// TIA Portal V18 export
FUNCTION "SS1_A6_16DI_IO_Update" : Void   // FC11060, LAD
{ S7_Optimized_Access := 'TRUE' }
VERSION : 0.1
// stored: AutoNumber false, IsIECCheckEnabled false, SetENOAutomatically false, UDAEnableTagReadback false
BEGIN

REGION Network 1: DIa0
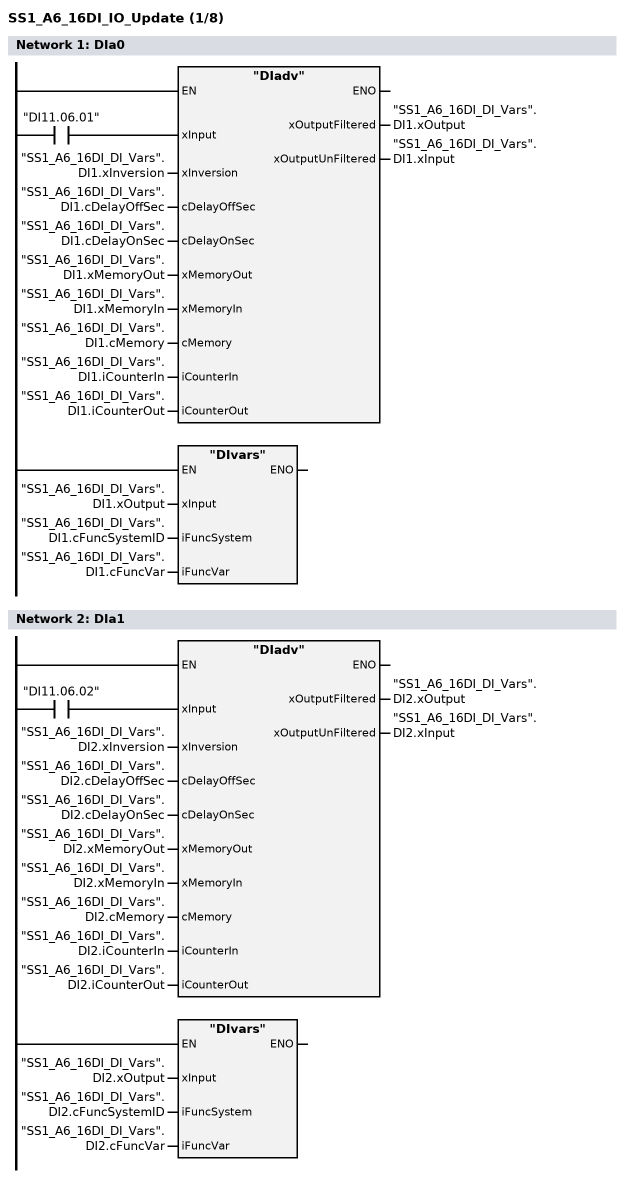
   RUNG wire#powerrail
      "DIadv"(xInput := wire#w1, xInversion := "SS1_A6_16DI_DI_Vars".DI1.xInversion, cDelayOffSec := "SS1_A6_16DI_DI_Vars".DI1.cDelayOffSec, cDelayOnSec := "SS1_A6_16DI_DI_Vars".DI1.cDelayOnSec, xMemoryOut := "SS1_A6_16DI_DI_Vars".DI1.xMemoryOut, xMemoryIn := "SS1_A6_16DI_DI_Vars".DI1.xMemoryIn, cMemory := "SS1_A6_16DI_DI_Vars".DI1.cMemory, xOutputFiltered => "SS1_A6_16DI_DI_Vars".DI1.xOutput, xOutputUnFiltered => "SS1_A6_16DI_DI_Vars".DI1.xInput, iCounterIn := "SS1_A6_16DI_DI_Vars".DI1.iCounterIn, iCounterOut := "SS1_A6_16DI_DI_Vars".DI1.iCounterOut)
   END_RUNG
   RUNG wire#powerrail
      Contact( "DI11.06.01" )
   END_RUNG wire#w1
   RUNG wire#powerrail
      "DIvars"(xInput := "SS1_A6_16DI_DI_Vars".DI1.xOutput, iFuncSystem := "SS1_A6_16DI_DI_Vars".DI1.cFuncSystemID, iFuncVar := "SS1_A6_16DI_DI_Vars".DI1.cFuncVar)
   END_RUNG
   // the same network as SCL:
   "DIadv"(xInput := "DI11.06.01",
           xInversion := "SS1_A6_16DI_DI_Vars".DI1.xInversion,
           cDelayOffSec := "SS1_A6_16DI_DI_Vars".DI1.cDelayOffSec,
           cDelayOnSec := "SS1_A6_16DI_DI_Vars".DI1.cDelayOnSec,
           xMemoryOut := "SS1_A6_16DI_DI_Vars".DI1.xMemoryOut,
           xMemoryIn := "SS1_A6_16DI_DI_Vars".DI1.xMemoryIn,
           cMemory := "SS1_A6_16DI_DI_Vars".DI1.cMemory,
           iCounterIn := "SS1_A6_16DI_DI_Vars".DI1.iCounterIn,
           iCounterOut := "SS1_A6_16DI_DI_Vars".DI1.iCounterOut,
           xOutputFiltered => "SS1_A6_16DI_DI_Vars".DI1.xOutput,
           xOutputUnFiltered => "SS1_A6_16DI_DI_Vars".DI1.xInput);
   "DIvars"(xInput := "SS1_A6_16DI_DI_Vars".DI1.xOutput,
            iFuncSystem := "SS1_A6_16DI_DI_Vars".DI1.cFuncSystemID,
            iFuncVar := "SS1_A6_16DI_DI_Vars".DI1.cFuncVar);
END_REGION

REGION Network 2: DIa1
   RUNG wire#powerrail
      "DIadv"(xInput := wire#w1, xInversion := "SS1_A6_16DI_DI_Vars".DI2.xInversion, cDelayOffSec := "SS1_A6_16DI_DI_Vars".DI2.cDelayOffSec, cDelayOnSec := "SS1_A6_16DI_DI_Vars".DI2.cDelayOnSec, xMemoryOut := "SS1_A6_16DI_DI_Vars".DI2.xMemoryOut, xMemoryIn := "SS1_A6_16DI_DI_Vars".DI2.xMemoryIn, cMemory := "SS1_A6_16DI_DI_Vars".DI2.cMemory, xOutputFiltered => "SS1_A6_16DI_DI_Vars".DI2.xOutput, xOutputUnFiltered => "SS1_A6_16DI_DI_Vars".DI2.xInput, iCounterIn := "SS1_A6_16DI_DI_Vars".DI2.iCounterIn, iCounterOut := "SS1_A6_16DI_DI_Vars".DI2.iCounterOut)
   END_RUNG
   RUNG wire#powerrail
      Contact( "DI11.06.02" )
   END_RUNG wire#w1
   RUNG wire#powerrail
      "DIvars"(xInput := "SS1_A6_16DI_DI_Vars".DI2.xOutput, iFuncSystem := "SS1_A6_16DI_DI_Vars".DI2.cFuncSystemID, iFuncVar := "SS1_A6_16DI_DI_Vars".DI2.cFuncVar)
   END_RUNG
   // the same network as SCL:
   "DIadv"(xInput := "DI11.06.02",
           xInversion := "SS1_A6_16DI_DI_Vars".DI2.xInversion,
           cDelayOffSec := "SS1_A6_16DI_DI_Vars".DI2.cDelayOffSec,
           cDelayOnSec := "SS1_A6_16DI_DI_Vars".DI2.cDelayOnSec,
           xMemoryOut := "SS1_A6_16DI_DI_Vars".DI2.xMemoryOut,
           xMemoryIn := "SS1_A6_16DI_DI_Vars".DI2.xMemoryIn,
           cMemory := "SS1_A6_16DI_DI_Vars".DI2.cMemory,
           iCounterIn := "SS1_A6_16DI_DI_Vars".DI2.iCounterIn,
           iCounterOut := "SS1_A6_16DI_DI_Vars".DI2.iCounterOut,
           xOutputFiltered => "SS1_A6_16DI_DI_Vars".DI2.xOutput,
           xOutputUnFiltered => "SS1_A6_16DI_DI_Vars".DI2.xInput);
   "DIvars"(xInput := "SS1_A6_16DI_DI_Vars".DI2.xOutput,
            iFuncSystem := "SS1_A6_16DI_DI_Vars".DI2.cFuncSystemID,
            iFuncVar := "SS1_A6_16DI_DI_Vars".DI2.cFuncVar);
END_REGION

REGION Network 3: DIa2
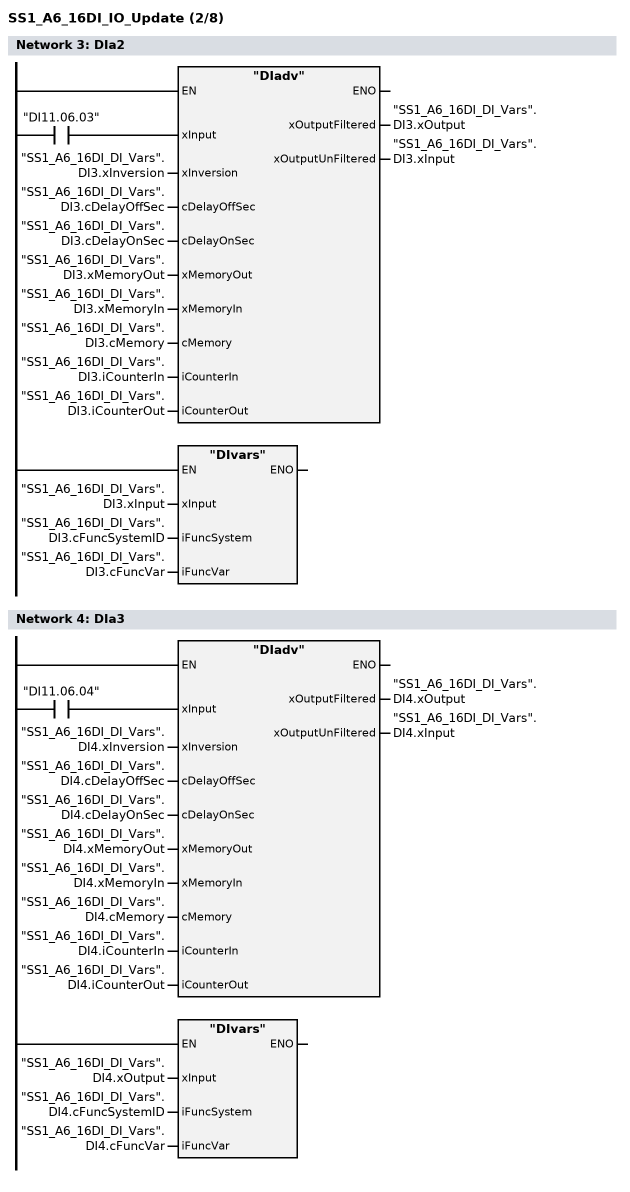
   RUNG wire#powerrail
      "DIadv"(xInput := wire#w1, xInversion := "SS1_A6_16DI_DI_Vars".DI3.xInversion, cDelayOffSec := "SS1_A6_16DI_DI_Vars".DI3.cDelayOffSec, cDelayOnSec := "SS1_A6_16DI_DI_Vars".DI3.cDelayOnSec, xMemoryOut := "SS1_A6_16DI_DI_Vars".DI3.xMemoryOut, xMemoryIn := "SS1_A6_16DI_DI_Vars".DI3.xMemoryIn, cMemory := "SS1_A6_16DI_DI_Vars".DI3.cMemory, xOutputFiltered => "SS1_A6_16DI_DI_Vars".DI3.xOutput, xOutputUnFiltered => "SS1_A6_16DI_DI_Vars".DI3.xInput, iCounterIn := "SS1_A6_16DI_DI_Vars".DI3.iCounterIn, iCounterOut := "SS1_A6_16DI_DI_Vars".DI3.iCounterOut)
   END_RUNG
   RUNG wire#powerrail
      Contact( "DI11.06.03" )
   END_RUNG wire#w1
   RUNG wire#powerrail
      "DIvars"(xInput := "SS1_A6_16DI_DI_Vars".DI3.xInput, iFuncSystem := "SS1_A6_16DI_DI_Vars".DI3.cFuncSystemID, iFuncVar := "SS1_A6_16DI_DI_Vars".DI3.cFuncVar)
   END_RUNG
   // the same network as SCL:
   "DIadv"(xInput := "DI11.06.03",
           xInversion := "SS1_A6_16DI_DI_Vars".DI3.xInversion,
           cDelayOffSec := "SS1_A6_16DI_DI_Vars".DI3.cDelayOffSec,
           cDelayOnSec := "SS1_A6_16DI_DI_Vars".DI3.cDelayOnSec,
           xMemoryOut := "SS1_A6_16DI_DI_Vars".DI3.xMemoryOut,
           xMemoryIn := "SS1_A6_16DI_DI_Vars".DI3.xMemoryIn,
           cMemory := "SS1_A6_16DI_DI_Vars".DI3.cMemory,
           iCounterIn := "SS1_A6_16DI_DI_Vars".DI3.iCounterIn,
           iCounterOut := "SS1_A6_16DI_DI_Vars".DI3.iCounterOut,
           xOutputFiltered => "SS1_A6_16DI_DI_Vars".DI3.xOutput,
           xOutputUnFiltered => "SS1_A6_16DI_DI_Vars".DI3.xInput);
   "DIvars"(xInput := "SS1_A6_16DI_DI_Vars".DI3.xInput,
            iFuncSystem := "SS1_A6_16DI_DI_Vars".DI3.cFuncSystemID,
            iFuncVar := "SS1_A6_16DI_DI_Vars".DI3.cFuncVar);
END_REGION

REGION Network 4: DIa3
   RUNG wire#powerrail
      "DIadv"(xInput := wire#w1, xInversion := "SS1_A6_16DI_DI_Vars".DI4.xInversion, cDelayOffSec := "SS1_A6_16DI_DI_Vars".DI4.cDelayOffSec, cDelayOnSec := "SS1_A6_16DI_DI_Vars".DI4.cDelayOnSec, xMemoryOut := "SS1_A6_16DI_DI_Vars".DI4.xMemoryOut, xMemoryIn := "SS1_A6_16DI_DI_Vars".DI4.xMemoryIn, cMemory := "SS1_A6_16DI_DI_Vars".DI4.cMemory, xOutputFiltered => "SS1_A6_16DI_DI_Vars".DI4.xOutput, xOutputUnFiltered => "SS1_A6_16DI_DI_Vars".DI4.xInput, iCounterIn := "SS1_A6_16DI_DI_Vars".DI4.iCounterIn, iCounterOut := "SS1_A6_16DI_DI_Vars".DI4.iCounterOut)
   END_RUNG
   RUNG wire#powerrail
      Contact( "DI11.06.04" )
   END_RUNG wire#w1
   RUNG wire#powerrail
      "DIvars"(xInput := "SS1_A6_16DI_DI_Vars".DI4.xOutput, iFuncSystem := "SS1_A6_16DI_DI_Vars".DI4.cFuncSystemID, iFuncVar := "SS1_A6_16DI_DI_Vars".DI4.cFuncVar)
   END_RUNG
   // the same network as SCL:
   "DIadv"(xInput := "DI11.06.04",
           xInversion := "SS1_A6_16DI_DI_Vars".DI4.xInversion,
           cDelayOffSec := "SS1_A6_16DI_DI_Vars".DI4.cDelayOffSec,
           cDelayOnSec := "SS1_A6_16DI_DI_Vars".DI4.cDelayOnSec,
           xMemoryOut := "SS1_A6_16DI_DI_Vars".DI4.xMemoryOut,
           xMemoryIn := "SS1_A6_16DI_DI_Vars".DI4.xMemoryIn,
           cMemory := "SS1_A6_16DI_DI_Vars".DI4.cMemory,
           iCounterIn := "SS1_A6_16DI_DI_Vars".DI4.iCounterIn,
           iCounterOut := "SS1_A6_16DI_DI_Vars".DI4.iCounterOut,
           xOutputFiltered => "SS1_A6_16DI_DI_Vars".DI4.xOutput,
           xOutputUnFiltered => "SS1_A6_16DI_DI_Vars".DI4.xInput);
   "DIvars"(xInput := "SS1_A6_16DI_DI_Vars".DI4.xOutput,
            iFuncSystem := "SS1_A6_16DI_DI_Vars".DI4.cFuncSystemID,
            iFuncVar := "SS1_A6_16DI_DI_Vars".DI4.cFuncVar);
END_REGION

REGION Network 5: DIa4
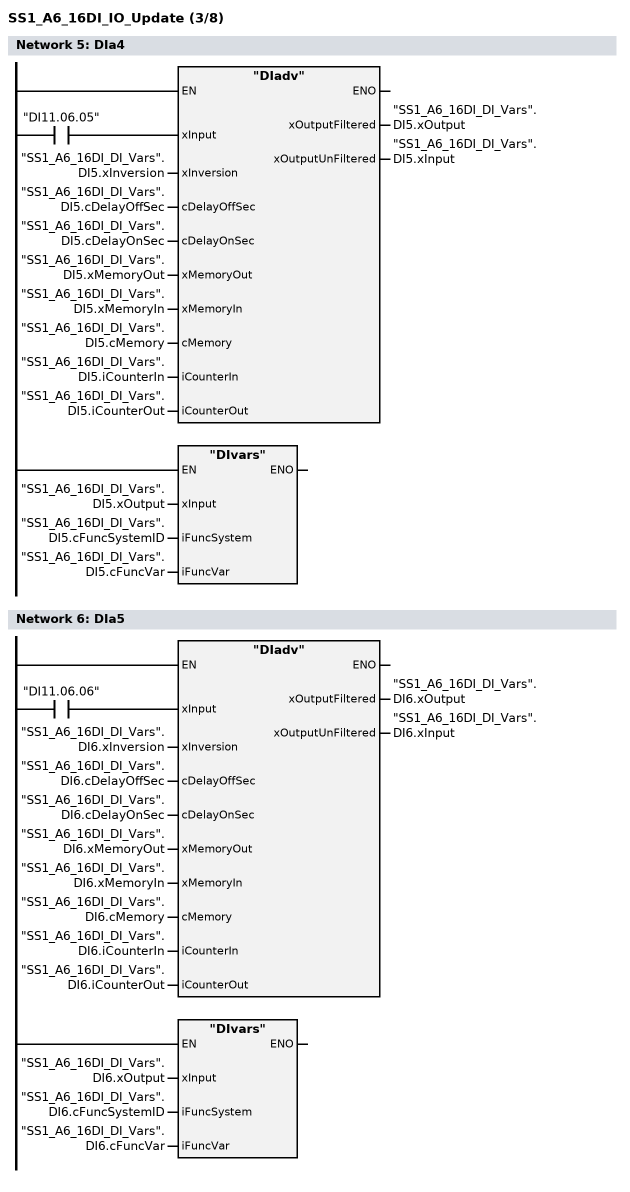
   RUNG wire#powerrail
      "DIadv"(xInput := wire#w1, xInversion := "SS1_A6_16DI_DI_Vars".DI5.xInversion, cDelayOffSec := "SS1_A6_16DI_DI_Vars".DI5.cDelayOffSec, cDelayOnSec := "SS1_A6_16DI_DI_Vars".DI5.cDelayOnSec, xMemoryOut := "SS1_A6_16DI_DI_Vars".DI5.xMemoryOut, xMemoryIn := "SS1_A6_16DI_DI_Vars".DI5.xMemoryIn, cMemory := "SS1_A6_16DI_DI_Vars".DI5.cMemory, xOutputFiltered => "SS1_A6_16DI_DI_Vars".DI5.xOutput, xOutputUnFiltered => "SS1_A6_16DI_DI_Vars".DI5.xInput, iCounterIn := "SS1_A6_16DI_DI_Vars".DI5.iCounterIn, iCounterOut := "SS1_A6_16DI_DI_Vars".DI5.iCounterOut)
   END_RUNG
   RUNG wire#powerrail
      Contact( "DI11.06.05" )
   END_RUNG wire#w1
   RUNG wire#powerrail
      "DIvars"(xInput := "SS1_A6_16DI_DI_Vars".DI5.xOutput, iFuncSystem := "SS1_A6_16DI_DI_Vars".DI5.cFuncSystemID, iFuncVar := "SS1_A6_16DI_DI_Vars".DI5.cFuncVar)
   END_RUNG
   // the same network as SCL:
   "DIadv"(xInput := "DI11.06.05",
           xInversion := "SS1_A6_16DI_DI_Vars".DI5.xInversion,
           cDelayOffSec := "SS1_A6_16DI_DI_Vars".DI5.cDelayOffSec,
           cDelayOnSec := "SS1_A6_16DI_DI_Vars".DI5.cDelayOnSec,
           xMemoryOut := "SS1_A6_16DI_DI_Vars".DI5.xMemoryOut,
           xMemoryIn := "SS1_A6_16DI_DI_Vars".DI5.xMemoryIn,
           cMemory := "SS1_A6_16DI_DI_Vars".DI5.cMemory,
           iCounterIn := "SS1_A6_16DI_DI_Vars".DI5.iCounterIn,
           iCounterOut := "SS1_A6_16DI_DI_Vars".DI5.iCounterOut,
           xOutputFiltered => "SS1_A6_16DI_DI_Vars".DI5.xOutput,
           xOutputUnFiltered => "SS1_A6_16DI_DI_Vars".DI5.xInput);
   "DIvars"(xInput := "SS1_A6_16DI_DI_Vars".DI5.xOutput,
            iFuncSystem := "SS1_A6_16DI_DI_Vars".DI5.cFuncSystemID,
            iFuncVar := "SS1_A6_16DI_DI_Vars".DI5.cFuncVar);
END_REGION

REGION Network 6: DIa5
   RUNG wire#powerrail
      "DIadv"(xInput := wire#w1, xInversion := "SS1_A6_16DI_DI_Vars".DI6.xInversion, cDelayOffSec := "SS1_A6_16DI_DI_Vars".DI6.cDelayOffSec, cDelayOnSec := "SS1_A6_16DI_DI_Vars".DI6.cDelayOnSec, xMemoryOut := "SS1_A6_16DI_DI_Vars".DI6.xMemoryOut, xMemoryIn := "SS1_A6_16DI_DI_Vars".DI6.xMemoryIn, cMemory := "SS1_A6_16DI_DI_Vars".DI6.cMemory, xOutputFiltered => "SS1_A6_16DI_DI_Vars".DI6.xOutput, xOutputUnFiltered => "SS1_A6_16DI_DI_Vars".DI6.xInput, iCounterIn := "SS1_A6_16DI_DI_Vars".DI6.iCounterIn, iCounterOut := "SS1_A6_16DI_DI_Vars".DI6.iCounterOut)
   END_RUNG
   RUNG wire#powerrail
      Contact( "DI11.06.06" )
   END_RUNG wire#w1
   RUNG wire#powerrail
      "DIvars"(xInput := "SS1_A6_16DI_DI_Vars".DI6.xOutput, iFuncSystem := "SS1_A6_16DI_DI_Vars".DI6.cFuncSystemID, iFuncVar := "SS1_A6_16DI_DI_Vars".DI6.cFuncVar)
   END_RUNG
   // the same network as SCL:
   "DIadv"(xInput := "DI11.06.06",
           xInversion := "SS1_A6_16DI_DI_Vars".DI6.xInversion,
           cDelayOffSec := "SS1_A6_16DI_DI_Vars".DI6.cDelayOffSec,
           cDelayOnSec := "SS1_A6_16DI_DI_Vars".DI6.cDelayOnSec,
           xMemoryOut := "SS1_A6_16DI_DI_Vars".DI6.xMemoryOut,
           xMemoryIn := "SS1_A6_16DI_DI_Vars".DI6.xMemoryIn,
           cMemory := "SS1_A6_16DI_DI_Vars".DI6.cMemory,
           iCounterIn := "SS1_A6_16DI_DI_Vars".DI6.iCounterIn,
           iCounterOut := "SS1_A6_16DI_DI_Vars".DI6.iCounterOut,
           xOutputFiltered => "SS1_A6_16DI_DI_Vars".DI6.xOutput,
           xOutputUnFiltered => "SS1_A6_16DI_DI_Vars".DI6.xInput);
   "DIvars"(xInput := "SS1_A6_16DI_DI_Vars".DI6.xOutput,
            iFuncSystem := "SS1_A6_16DI_DI_Vars".DI6.cFuncSystemID,
            iFuncVar := "SS1_A6_16DI_DI_Vars".DI6.cFuncVar);
END_REGION

REGION Network 7: DIa6
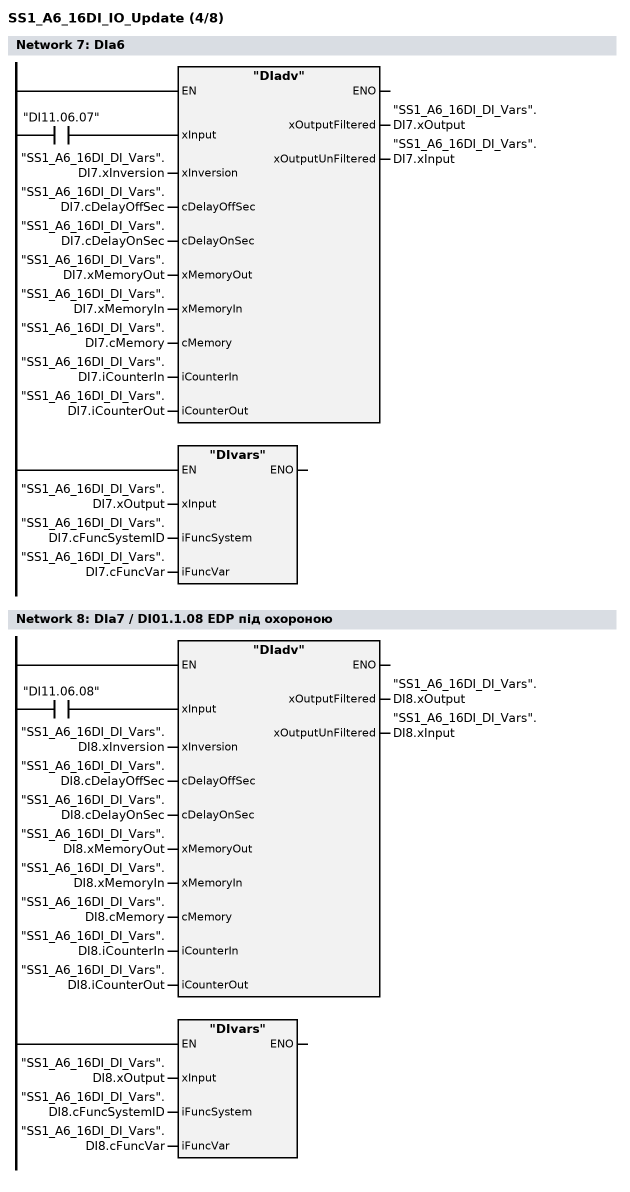
   RUNG wire#powerrail
      "DIadv"(xInput := wire#w1, xInversion := "SS1_A6_16DI_DI_Vars".DI7.xInversion, cDelayOffSec := "SS1_A6_16DI_DI_Vars".DI7.cDelayOffSec, cDelayOnSec := "SS1_A6_16DI_DI_Vars".DI7.cDelayOnSec, xMemoryOut := "SS1_A6_16DI_DI_Vars".DI7.xMemoryOut, xMemoryIn := "SS1_A6_16DI_DI_Vars".DI7.xMemoryIn, cMemory := "SS1_A6_16DI_DI_Vars".DI7.cMemory, xOutputFiltered => "SS1_A6_16DI_DI_Vars".DI7.xOutput, xOutputUnFiltered => "SS1_A6_16DI_DI_Vars".DI7.xInput, iCounterIn := "SS1_A6_16DI_DI_Vars".DI7.iCounterIn, iCounterOut := "SS1_A6_16DI_DI_Vars".DI7.iCounterOut)
   END_RUNG
   RUNG wire#powerrail
      Contact( "DI11.06.07" )
   END_RUNG wire#w1
   RUNG wire#powerrail
      "DIvars"(xInput := "SS1_A6_16DI_DI_Vars".DI7.xOutput, iFuncSystem := "SS1_A6_16DI_DI_Vars".DI7.cFuncSystemID, iFuncVar := "SS1_A6_16DI_DI_Vars".DI7.cFuncVar)
   END_RUNG
   // the same network as SCL:
   "DIadv"(xInput := "DI11.06.07",
           xInversion := "SS1_A6_16DI_DI_Vars".DI7.xInversion,
           cDelayOffSec := "SS1_A6_16DI_DI_Vars".DI7.cDelayOffSec,
           cDelayOnSec := "SS1_A6_16DI_DI_Vars".DI7.cDelayOnSec,
           xMemoryOut := "SS1_A6_16DI_DI_Vars".DI7.xMemoryOut,
           xMemoryIn := "SS1_A6_16DI_DI_Vars".DI7.xMemoryIn,
           cMemory := "SS1_A6_16DI_DI_Vars".DI7.cMemory,
           iCounterIn := "SS1_A6_16DI_DI_Vars".DI7.iCounterIn,
           iCounterOut := "SS1_A6_16DI_DI_Vars".DI7.iCounterOut,
           xOutputFiltered => "SS1_A6_16DI_DI_Vars".DI7.xOutput,
           xOutputUnFiltered => "SS1_A6_16DI_DI_Vars".DI7.xInput);
   "DIvars"(xInput := "SS1_A6_16DI_DI_Vars".DI7.xOutput,
            iFuncSystem := "SS1_A6_16DI_DI_Vars".DI7.cFuncSystemID,
            iFuncVar := "SS1_A6_16DI_DI_Vars".DI7.cFuncVar);
END_REGION

REGION Network 8: DIa7 / DI01.1.08 EDP під охороною
   RUNG wire#powerrail
      "DIadv"(xInput := wire#w1, xInversion := "SS1_A6_16DI_DI_Vars".DI8.xInversion, cDelayOffSec := "SS1_A6_16DI_DI_Vars".DI8.cDelayOffSec, cDelayOnSec := "SS1_A6_16DI_DI_Vars".DI8.cDelayOnSec, xMemoryOut := "SS1_A6_16DI_DI_Vars".DI8.xMemoryOut, xMemoryIn := "SS1_A6_16DI_DI_Vars".DI8.xMemoryIn, cMemory := "SS1_A6_16DI_DI_Vars".DI8.cMemory, xOutputFiltered => "SS1_A6_16DI_DI_Vars".DI8.xOutput, xOutputUnFiltered => "SS1_A6_16DI_DI_Vars".DI8.xInput, iCounterIn := "SS1_A6_16DI_DI_Vars".DI8.iCounterIn, iCounterOut := "SS1_A6_16DI_DI_Vars".DI8.iCounterOut)
   END_RUNG
   RUNG wire#powerrail
      Contact( "DI11.06.08" )
   END_RUNG wire#w1
   RUNG wire#powerrail
      "DIvars"(xInput := "SS1_A6_16DI_DI_Vars".DI8.xOutput, iFuncSystem := "SS1_A6_16DI_DI_Vars".DI8.cFuncSystemID, iFuncVar := "SS1_A6_16DI_DI_Vars".DI8.cFuncVar)
   END_RUNG
   // the same network as SCL:
   "DIadv"(xInput := "DI11.06.08",
           xInversion := "SS1_A6_16DI_DI_Vars".DI8.xInversion,
           cDelayOffSec := "SS1_A6_16DI_DI_Vars".DI8.cDelayOffSec,
           cDelayOnSec := "SS1_A6_16DI_DI_Vars".DI8.cDelayOnSec,
           xMemoryOut := "SS1_A6_16DI_DI_Vars".DI8.xMemoryOut,
           xMemoryIn := "SS1_A6_16DI_DI_Vars".DI8.xMemoryIn,
           cMemory := "SS1_A6_16DI_DI_Vars".DI8.cMemory,
           iCounterIn := "SS1_A6_16DI_DI_Vars".DI8.iCounterIn,
           iCounterOut := "SS1_A6_16DI_DI_Vars".DI8.iCounterOut,
           xOutputFiltered => "SS1_A6_16DI_DI_Vars".DI8.xOutput,
           xOutputUnFiltered => "SS1_A6_16DI_DI_Vars".DI8.xInput);
   "DIvars"(xInput := "SS1_A6_16DI_DI_Vars".DI8.xOutput,
            iFuncSystem := "SS1_A6_16DI_DI_Vars".DI8.cFuncSystemID,
            iFuncVar := "SS1_A6_16DI_DI_Vars".DI8.cFuncVar);
END_REGION

REGION Network 9: DIb0
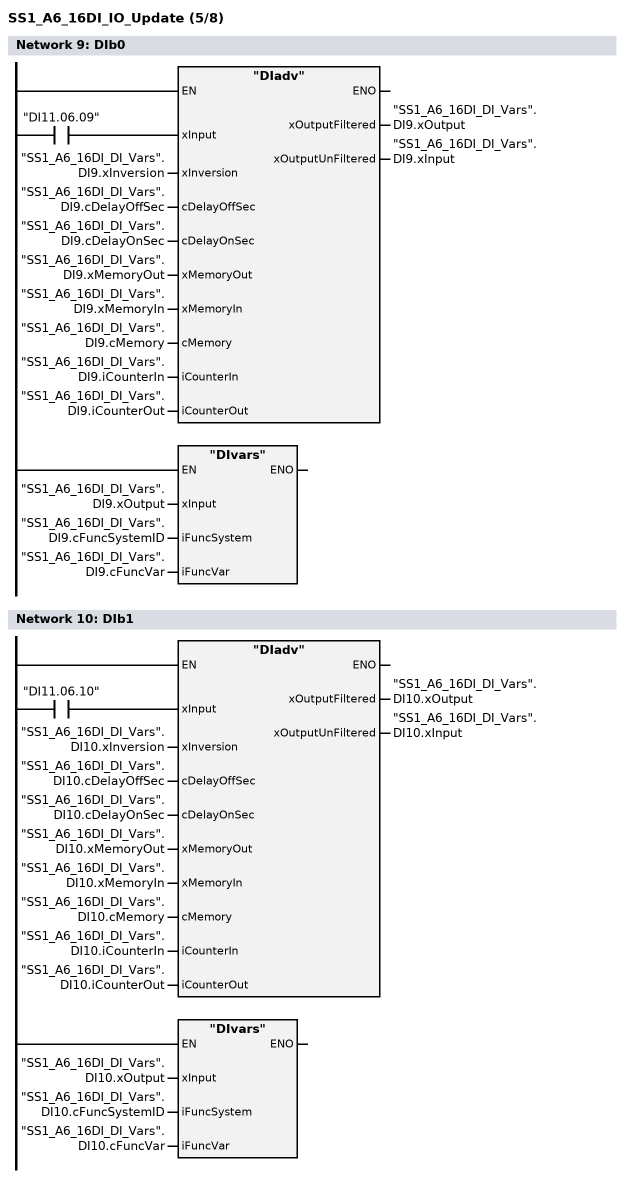
   RUNG wire#powerrail
      "DIadv"(xInput := wire#w1, xInversion := "SS1_A6_16DI_DI_Vars".DI9.xInversion, cDelayOffSec := "SS1_A6_16DI_DI_Vars".DI9.cDelayOffSec, cDelayOnSec := "SS1_A6_16DI_DI_Vars".DI9.cDelayOnSec, xMemoryOut := "SS1_A6_16DI_DI_Vars".DI9.xMemoryOut, xMemoryIn := "SS1_A6_16DI_DI_Vars".DI9.xMemoryIn, cMemory := "SS1_A6_16DI_DI_Vars".DI9.cMemory, iCounterIn := "SS1_A6_16DI_DI_Vars".DI9.iCounterIn, iCounterOut := "SS1_A6_16DI_DI_Vars".DI9.iCounterOut, xOutputFiltered => "SS1_A6_16DI_DI_Vars".DI9.xOutput, xOutputUnFiltered => "SS1_A6_16DI_DI_Vars".DI9.xInput)
   END_RUNG
   RUNG wire#powerrail
      Contact( "DI11.06.09" )
   END_RUNG wire#w1
   RUNG wire#powerrail
      "DIvars"(xInput := "SS1_A6_16DI_DI_Vars".DI9.xOutput, iFuncSystem := "SS1_A6_16DI_DI_Vars".DI9.cFuncSystemID, iFuncVar := "SS1_A6_16DI_DI_Vars".DI9.cFuncVar)
   END_RUNG
   // the same network as SCL:
   "DIadv"(xInput := "DI11.06.09",
           xInversion := "SS1_A6_16DI_DI_Vars".DI9.xInversion,
           cDelayOffSec := "SS1_A6_16DI_DI_Vars".DI9.cDelayOffSec,
           cDelayOnSec := "SS1_A6_16DI_DI_Vars".DI9.cDelayOnSec,
           xMemoryOut := "SS1_A6_16DI_DI_Vars".DI9.xMemoryOut,
           xMemoryIn := "SS1_A6_16DI_DI_Vars".DI9.xMemoryIn,
           cMemory := "SS1_A6_16DI_DI_Vars".DI9.cMemory,
           iCounterIn := "SS1_A6_16DI_DI_Vars".DI9.iCounterIn,
           iCounterOut := "SS1_A6_16DI_DI_Vars".DI9.iCounterOut,
           xOutputFiltered => "SS1_A6_16DI_DI_Vars".DI9.xOutput,
           xOutputUnFiltered => "SS1_A6_16DI_DI_Vars".DI9.xInput);
   "DIvars"(xInput := "SS1_A6_16DI_DI_Vars".DI9.xOutput,
            iFuncSystem := "SS1_A6_16DI_DI_Vars".DI9.cFuncSystemID,
            iFuncVar := "SS1_A6_16DI_DI_Vars".DI9.cFuncVar);
END_REGION

REGION Network 10: DIb1
   RUNG wire#powerrail
      "DIadv"(xInput := wire#w1, xInversion := "SS1_A6_16DI_DI_Vars".DI10.xInversion, cDelayOffSec := "SS1_A6_16DI_DI_Vars".DI10.cDelayOffSec, cDelayOnSec := "SS1_A6_16DI_DI_Vars".DI10.cDelayOnSec, xMemoryOut := "SS1_A6_16DI_DI_Vars".DI10.xMemoryOut, xMemoryIn := "SS1_A6_16DI_DI_Vars".DI10.xMemoryIn, cMemory := "SS1_A6_16DI_DI_Vars".DI10.cMemory, iCounterIn := "SS1_A6_16DI_DI_Vars".DI10.iCounterIn, iCounterOut := "SS1_A6_16DI_DI_Vars".DI10.iCounterOut, xOutputFiltered => "SS1_A6_16DI_DI_Vars".DI10.xOutput, xOutputUnFiltered => "SS1_A6_16DI_DI_Vars".DI10.xInput)
   END_RUNG
   RUNG wire#powerrail
      Contact( "DI11.06.10" )
   END_RUNG wire#w1
   RUNG wire#powerrail
      "DIvars"(xInput := "SS1_A6_16DI_DI_Vars".DI10.xOutput, iFuncSystem := "SS1_A6_16DI_DI_Vars".DI10.cFuncSystemID, iFuncVar := "SS1_A6_16DI_DI_Vars".DI10.cFuncVar)
   END_RUNG
   // the same network as SCL:
   "DIadv"(xInput := "DI11.06.10",
           xInversion := "SS1_A6_16DI_DI_Vars".DI10.xInversion,
           cDelayOffSec := "SS1_A6_16DI_DI_Vars".DI10.cDelayOffSec,
           cDelayOnSec := "SS1_A6_16DI_DI_Vars".DI10.cDelayOnSec,
           xMemoryOut := "SS1_A6_16DI_DI_Vars".DI10.xMemoryOut,
           xMemoryIn := "SS1_A6_16DI_DI_Vars".DI10.xMemoryIn,
           cMemory := "SS1_A6_16DI_DI_Vars".DI10.cMemory,
           iCounterIn := "SS1_A6_16DI_DI_Vars".DI10.iCounterIn,
           iCounterOut := "SS1_A6_16DI_DI_Vars".DI10.iCounterOut,
           xOutputFiltered => "SS1_A6_16DI_DI_Vars".DI10.xOutput,
           xOutputUnFiltered => "SS1_A6_16DI_DI_Vars".DI10.xInput);
   "DIvars"(xInput := "SS1_A6_16DI_DI_Vars".DI10.xOutput,
            iFuncSystem := "SS1_A6_16DI_DI_Vars".DI10.cFuncSystemID,
            iFuncVar := "SS1_A6_16DI_DI_Vars".DI10.cFuncVar);
END_REGION

REGION Network 11: DIb2
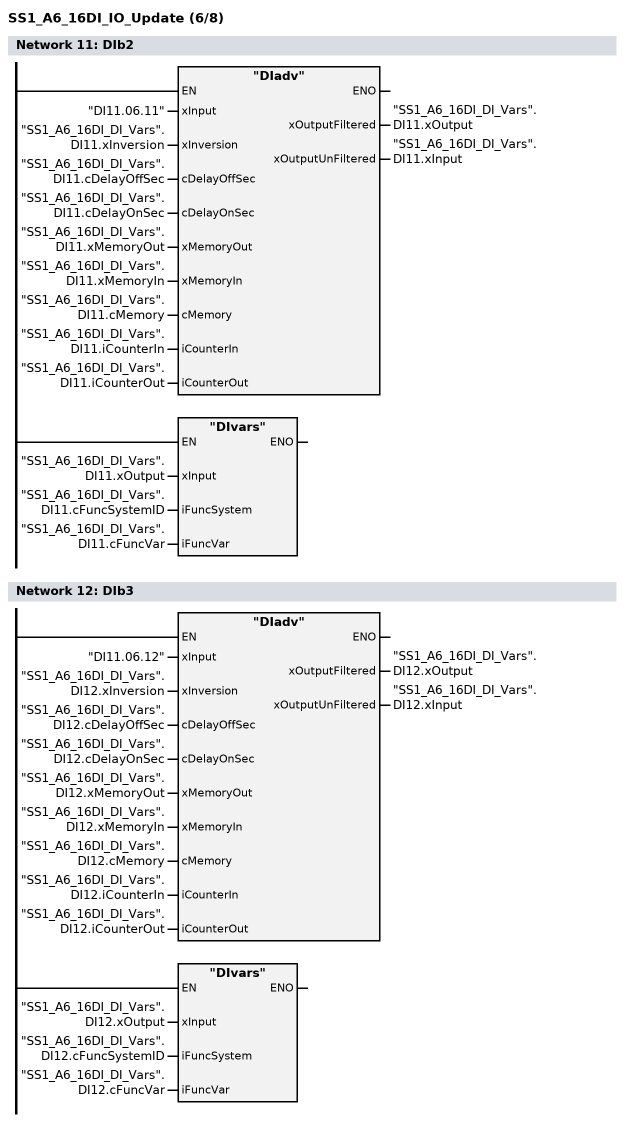
   RUNG wire#powerrail
      "DIadv"(xInput := "DI11.06.11", xInversion := "SS1_A6_16DI_DI_Vars".DI11.xInversion, cDelayOffSec := "SS1_A6_16DI_DI_Vars".DI11.cDelayOffSec, cDelayOnSec := "SS1_A6_16DI_DI_Vars".DI11.cDelayOnSec, xMemoryOut := "SS1_A6_16DI_DI_Vars".DI11.xMemoryOut, xMemoryIn := "SS1_A6_16DI_DI_Vars".DI11.xMemoryIn, cMemory := "SS1_A6_16DI_DI_Vars".DI11.cMemory, xOutputFiltered => "SS1_A6_16DI_DI_Vars".DI11.xOutput, xOutputUnFiltered => "SS1_A6_16DI_DI_Vars".DI11.xInput, iCounterIn := "SS1_A6_16DI_DI_Vars".DI11.iCounterIn, iCounterOut := "SS1_A6_16DI_DI_Vars".DI11.iCounterOut)
   END_RUNG
   RUNG wire#powerrail
      "DIvars"(xInput := "SS1_A6_16DI_DI_Vars".DI11.xOutput, iFuncSystem := "SS1_A6_16DI_DI_Vars".DI11.cFuncSystemID, iFuncVar := "SS1_A6_16DI_DI_Vars".DI11.cFuncVar)
   END_RUNG
   // the same network as SCL:
   "DIadv"(xInput := "DI11.06.11",
           xInversion := "SS1_A6_16DI_DI_Vars".DI11.xInversion,
           cDelayOffSec := "SS1_A6_16DI_DI_Vars".DI11.cDelayOffSec,
           cDelayOnSec := "SS1_A6_16DI_DI_Vars".DI11.cDelayOnSec,
           xMemoryOut := "SS1_A6_16DI_DI_Vars".DI11.xMemoryOut,
           xMemoryIn := "SS1_A6_16DI_DI_Vars".DI11.xMemoryIn,
           cMemory := "SS1_A6_16DI_DI_Vars".DI11.cMemory,
           iCounterIn := "SS1_A6_16DI_DI_Vars".DI11.iCounterIn,
           iCounterOut := "SS1_A6_16DI_DI_Vars".DI11.iCounterOut,
           xOutputFiltered => "SS1_A6_16DI_DI_Vars".DI11.xOutput,
           xOutputUnFiltered => "SS1_A6_16DI_DI_Vars".DI11.xInput);
   "DIvars"(xInput := "SS1_A6_16DI_DI_Vars".DI11.xOutput,
            iFuncSystem := "SS1_A6_16DI_DI_Vars".DI11.cFuncSystemID,
            iFuncVar := "SS1_A6_16DI_DI_Vars".DI11.cFuncVar);
END_REGION

REGION Network 12: DIb3
   RUNG wire#powerrail
      "DIadv"(xInput := "DI11.06.12", xInversion := "SS1_A6_16DI_DI_Vars".DI12.xInversion, cDelayOffSec := "SS1_A6_16DI_DI_Vars".DI12.cDelayOffSec, cDelayOnSec := "SS1_A6_16DI_DI_Vars".DI12.cDelayOnSec, xMemoryOut := "SS1_A6_16DI_DI_Vars".DI12.xMemoryOut, xMemoryIn := "SS1_A6_16DI_DI_Vars".DI12.xMemoryIn, cMemory := "SS1_A6_16DI_DI_Vars".DI12.cMemory, xOutputFiltered => "SS1_A6_16DI_DI_Vars".DI12.xOutput, xOutputUnFiltered => "SS1_A6_16DI_DI_Vars".DI12.xInput, iCounterIn := "SS1_A6_16DI_DI_Vars".DI12.iCounterIn, iCounterOut := "SS1_A6_16DI_DI_Vars".DI12.iCounterOut)
   END_RUNG
   RUNG wire#powerrail
      "DIvars"(xInput := "SS1_A6_16DI_DI_Vars".DI12.xOutput, iFuncSystem := "SS1_A6_16DI_DI_Vars".DI12.cFuncSystemID, iFuncVar := "SS1_A6_16DI_DI_Vars".DI12.cFuncVar)
   END_RUNG
   // the same network as SCL:
   "DIadv"(xInput := "DI11.06.12",
           xInversion := "SS1_A6_16DI_DI_Vars".DI12.xInversion,
           cDelayOffSec := "SS1_A6_16DI_DI_Vars".DI12.cDelayOffSec,
           cDelayOnSec := "SS1_A6_16DI_DI_Vars".DI12.cDelayOnSec,
           xMemoryOut := "SS1_A6_16DI_DI_Vars".DI12.xMemoryOut,
           xMemoryIn := "SS1_A6_16DI_DI_Vars".DI12.xMemoryIn,
           cMemory := "SS1_A6_16DI_DI_Vars".DI12.cMemory,
           iCounterIn := "SS1_A6_16DI_DI_Vars".DI12.iCounterIn,
           iCounterOut := "SS1_A6_16DI_DI_Vars".DI12.iCounterOut,
           xOutputFiltered => "SS1_A6_16DI_DI_Vars".DI12.xOutput,
           xOutputUnFiltered => "SS1_A6_16DI_DI_Vars".DI12.xInput);
   "DIvars"(xInput := "SS1_A6_16DI_DI_Vars".DI12.xOutput,
            iFuncSystem := "SS1_A6_16DI_DI_Vars".DI12.cFuncSystemID,
            iFuncVar := "SS1_A6_16DI_DI_Vars".DI12.cFuncVar);
END_REGION

REGION Network 13: DIb4
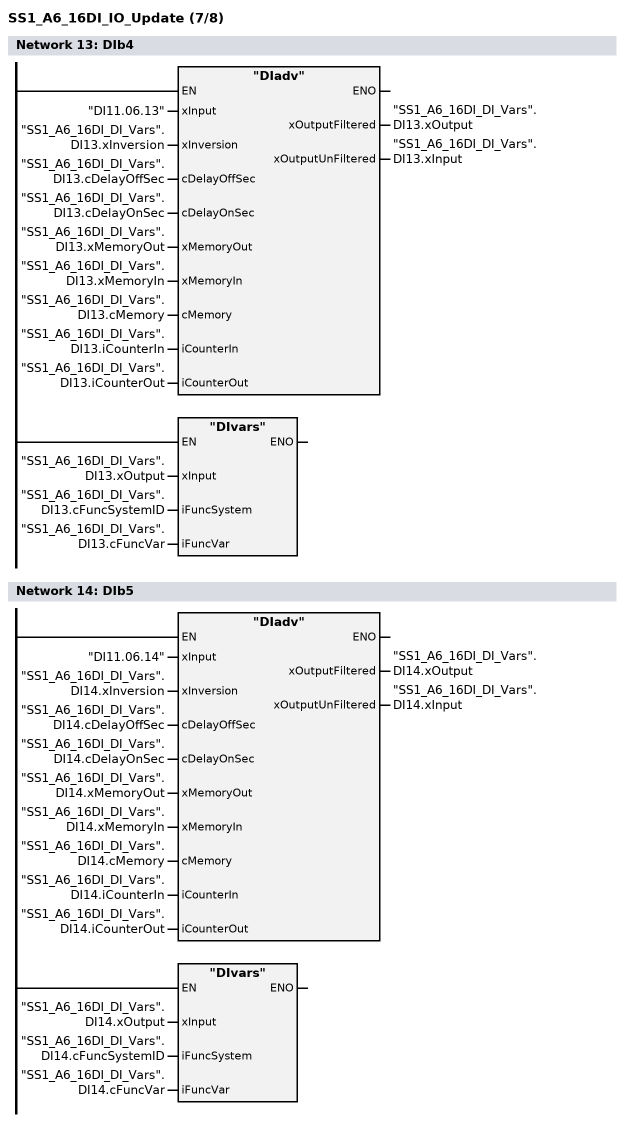
   RUNG wire#powerrail
      "DIadv"(xInput := "DI11.06.13", xInversion := "SS1_A6_16DI_DI_Vars".DI13.xInversion, cDelayOffSec := "SS1_A6_16DI_DI_Vars".DI13.cDelayOffSec, cDelayOnSec := "SS1_A6_16DI_DI_Vars".DI13.cDelayOnSec, xMemoryOut := "SS1_A6_16DI_DI_Vars".DI13.xMemoryOut, xMemoryIn := "SS1_A6_16DI_DI_Vars".DI13.xMemoryIn, cMemory := "SS1_A6_16DI_DI_Vars".DI13.cMemory, xOutputFiltered => "SS1_A6_16DI_DI_Vars".DI13.xOutput, xOutputUnFiltered => "SS1_A6_16DI_DI_Vars".DI13.xInput, iCounterIn := "SS1_A6_16DI_DI_Vars".DI13.iCounterIn, iCounterOut := "SS1_A6_16DI_DI_Vars".DI13.iCounterOut)
   END_RUNG
   RUNG wire#powerrail
      "DIvars"(xInput := "SS1_A6_16DI_DI_Vars".DI13.xOutput, iFuncSystem := "SS1_A6_16DI_DI_Vars".DI13.cFuncSystemID, iFuncVar := "SS1_A6_16DI_DI_Vars".DI13.cFuncVar)
   END_RUNG
   // the same network as SCL:
   "DIadv"(xInput := "DI11.06.13",
           xInversion := "SS1_A6_16DI_DI_Vars".DI13.xInversion,
           cDelayOffSec := "SS1_A6_16DI_DI_Vars".DI13.cDelayOffSec,
           cDelayOnSec := "SS1_A6_16DI_DI_Vars".DI13.cDelayOnSec,
           xMemoryOut := "SS1_A6_16DI_DI_Vars".DI13.xMemoryOut,
           xMemoryIn := "SS1_A6_16DI_DI_Vars".DI13.xMemoryIn,
           cMemory := "SS1_A6_16DI_DI_Vars".DI13.cMemory,
           iCounterIn := "SS1_A6_16DI_DI_Vars".DI13.iCounterIn,
           iCounterOut := "SS1_A6_16DI_DI_Vars".DI13.iCounterOut,
           xOutputFiltered => "SS1_A6_16DI_DI_Vars".DI13.xOutput,
           xOutputUnFiltered => "SS1_A6_16DI_DI_Vars".DI13.xInput);
   "DIvars"(xInput := "SS1_A6_16DI_DI_Vars".DI13.xOutput,
            iFuncSystem := "SS1_A6_16DI_DI_Vars".DI13.cFuncSystemID,
            iFuncVar := "SS1_A6_16DI_DI_Vars".DI13.cFuncVar);
END_REGION

REGION Network 14: DIb5
   RUNG wire#powerrail
      "DIadv"(xInput := "DI11.06.14", xInversion := "SS1_A6_16DI_DI_Vars".DI14.xInversion, cDelayOffSec := "SS1_A6_16DI_DI_Vars".DI14.cDelayOffSec, cDelayOnSec := "SS1_A6_16DI_DI_Vars".DI14.cDelayOnSec, xMemoryOut := "SS1_A6_16DI_DI_Vars".DI14.xMemoryOut, xMemoryIn := "SS1_A6_16DI_DI_Vars".DI14.xMemoryIn, cMemory := "SS1_A6_16DI_DI_Vars".DI14.cMemory, xOutputFiltered => "SS1_A6_16DI_DI_Vars".DI14.xOutput, xOutputUnFiltered => "SS1_A6_16DI_DI_Vars".DI14.xInput, iCounterIn := "SS1_A6_16DI_DI_Vars".DI14.iCounterIn, iCounterOut := "SS1_A6_16DI_DI_Vars".DI14.iCounterOut)
   END_RUNG
   RUNG wire#powerrail
      "DIvars"(xInput := "SS1_A6_16DI_DI_Vars".DI14.xOutput, iFuncSystem := "SS1_A6_16DI_DI_Vars".DI14.cFuncSystemID, iFuncVar := "SS1_A6_16DI_DI_Vars".DI14.cFuncVar)
   END_RUNG
   // the same network as SCL:
   "DIadv"(xInput := "DI11.06.14",
           xInversion := "SS1_A6_16DI_DI_Vars".DI14.xInversion,
           cDelayOffSec := "SS1_A6_16DI_DI_Vars".DI14.cDelayOffSec,
           cDelayOnSec := "SS1_A6_16DI_DI_Vars".DI14.cDelayOnSec,
           xMemoryOut := "SS1_A6_16DI_DI_Vars".DI14.xMemoryOut,
           xMemoryIn := "SS1_A6_16DI_DI_Vars".DI14.xMemoryIn,
           cMemory := "SS1_A6_16DI_DI_Vars".DI14.cMemory,
           iCounterIn := "SS1_A6_16DI_DI_Vars".DI14.iCounterIn,
           iCounterOut := "SS1_A6_16DI_DI_Vars".DI14.iCounterOut,
           xOutputFiltered => "SS1_A6_16DI_DI_Vars".DI14.xOutput,
           xOutputUnFiltered => "SS1_A6_16DI_DI_Vars".DI14.xInput);
   "DIvars"(xInput := "SS1_A6_16DI_DI_Vars".DI14.xOutput,
            iFuncSystem := "SS1_A6_16DI_DI_Vars".DI14.cFuncSystemID,
            iFuncVar := "SS1_A6_16DI_DI_Vars".DI14.cFuncVar);
END_REGION

REGION Network 15: DIb6
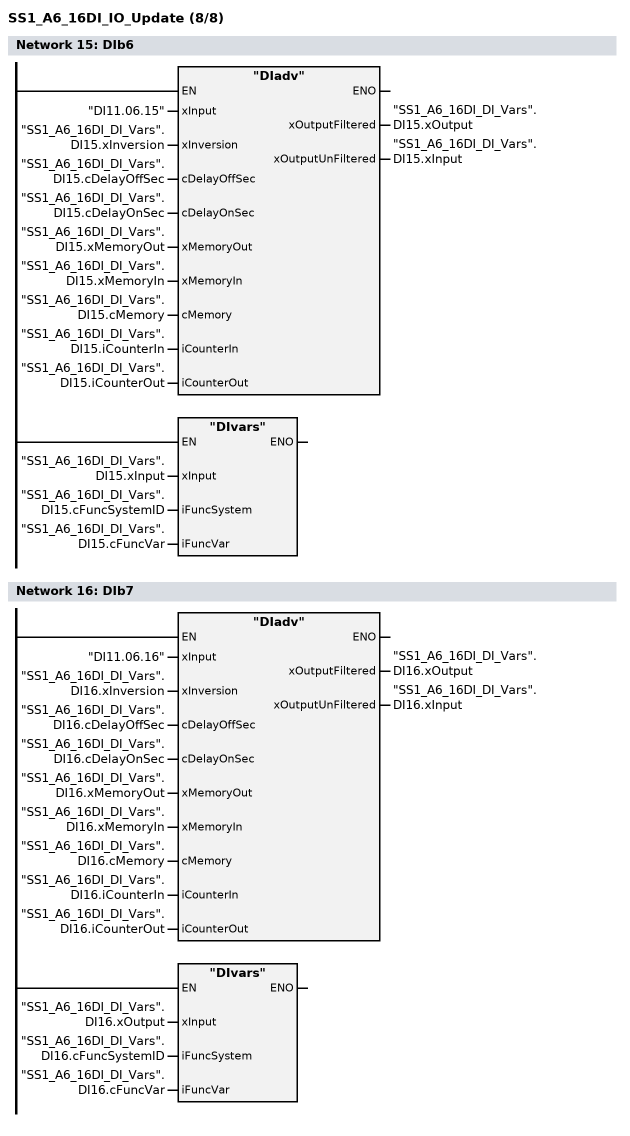
   RUNG wire#powerrail
      "DIadv"(xInput := "DI11.06.15", xInversion := "SS1_A6_16DI_DI_Vars".DI15.xInversion, cDelayOffSec := "SS1_A6_16DI_DI_Vars".DI15.cDelayOffSec, cDelayOnSec := "SS1_A6_16DI_DI_Vars".DI15.cDelayOnSec, xMemoryOut := "SS1_A6_16DI_DI_Vars".DI15.xMemoryOut, xMemoryIn := "SS1_A6_16DI_DI_Vars".DI15.xMemoryIn, cMemory := "SS1_A6_16DI_DI_Vars".DI15.cMemory, xOutputFiltered => "SS1_A6_16DI_DI_Vars".DI15.xOutput, xOutputUnFiltered => "SS1_A6_16DI_DI_Vars".DI15.xInput, iCounterIn := "SS1_A6_16DI_DI_Vars".DI15.iCounterIn, iCounterOut := "SS1_A6_16DI_DI_Vars".DI15.iCounterOut)
   END_RUNG
   RUNG wire#powerrail
      "DIvars"(xInput := "SS1_A6_16DI_DI_Vars".DI15.xInput, iFuncSystem := "SS1_A6_16DI_DI_Vars".DI15.cFuncSystemID, iFuncVar := "SS1_A6_16DI_DI_Vars".DI15.cFuncVar)
   END_RUNG
   // the same network as SCL:
   "DIadv"(xInput := "DI11.06.15",
           xInversion := "SS1_A6_16DI_DI_Vars".DI15.xInversion,
           cDelayOffSec := "SS1_A6_16DI_DI_Vars".DI15.cDelayOffSec,
           cDelayOnSec := "SS1_A6_16DI_DI_Vars".DI15.cDelayOnSec,
           xMemoryOut := "SS1_A6_16DI_DI_Vars".DI15.xMemoryOut,
           xMemoryIn := "SS1_A6_16DI_DI_Vars".DI15.xMemoryIn,
           cMemory := "SS1_A6_16DI_DI_Vars".DI15.cMemory,
           iCounterIn := "SS1_A6_16DI_DI_Vars".DI15.iCounterIn,
           iCounterOut := "SS1_A6_16DI_DI_Vars".DI15.iCounterOut,
           xOutputFiltered => "SS1_A6_16DI_DI_Vars".DI15.xOutput,
           xOutputUnFiltered => "SS1_A6_16DI_DI_Vars".DI15.xInput);
   "DIvars"(xInput := "SS1_A6_16DI_DI_Vars".DI15.xInput,
            iFuncSystem := "SS1_A6_16DI_DI_Vars".DI15.cFuncSystemID,
            iFuncVar := "SS1_A6_16DI_DI_Vars".DI15.cFuncVar);
END_REGION

REGION Network 16: DIb7
   RUNG wire#powerrail
      "DIadv"(xInput := "DI11.06.16", xInversion := "SS1_A6_16DI_DI_Vars".DI16.xInversion, cDelayOffSec := "SS1_A6_16DI_DI_Vars".DI16.cDelayOffSec, cDelayOnSec := "SS1_A6_16DI_DI_Vars".DI16.cDelayOnSec, xMemoryOut := "SS1_A6_16DI_DI_Vars".DI16.xMemoryOut, xMemoryIn := "SS1_A6_16DI_DI_Vars".DI16.xMemoryIn, cMemory := "SS1_A6_16DI_DI_Vars".DI16.cMemory, xOutputFiltered => "SS1_A6_16DI_DI_Vars".DI16.xOutput, xOutputUnFiltered => "SS1_A6_16DI_DI_Vars".DI16.xInput, iCounterIn := "SS1_A6_16DI_DI_Vars".DI16.iCounterIn, iCounterOut := "SS1_A6_16DI_DI_Vars".DI16.iCounterOut)
   END_RUNG
   RUNG wire#powerrail
      "DIvars"(xInput := "SS1_A6_16DI_DI_Vars".DI16.xOutput, iFuncSystem := "SS1_A6_16DI_DI_Vars".DI16.cFuncSystemID, iFuncVar := "SS1_A6_16DI_DI_Vars".DI16.cFuncVar)
   END_RUNG
   // the same network as SCL:
   "DIadv"(xInput := "DI11.06.16",
           xInversion := "SS1_A6_16DI_DI_Vars".DI16.xInversion,
           cDelayOffSec := "SS1_A6_16DI_DI_Vars".DI16.cDelayOffSec,
           cDelayOnSec := "SS1_A6_16DI_DI_Vars".DI16.cDelayOnSec,
           xMemoryOut := "SS1_A6_16DI_DI_Vars".DI16.xMemoryOut,
           xMemoryIn := "SS1_A6_16DI_DI_Vars".DI16.xMemoryIn,
           cMemory := "SS1_A6_16DI_DI_Vars".DI16.cMemory,
           iCounterIn := "SS1_A6_16DI_DI_Vars".DI16.iCounterIn,
           iCounterOut := "SS1_A6_16DI_DI_Vars".DI16.iCounterOut,
           xOutputFiltered => "SS1_A6_16DI_DI_Vars".DI16.xOutput,
           xOutputUnFiltered => "SS1_A6_16DI_DI_Vars".DI16.xInput);
   "DIvars"(xInput := "SS1_A6_16DI_DI_Vars".DI16.xOutput,
            iFuncSystem := "SS1_A6_16DI_DI_Vars".DI16.cFuncSystemID,
            iFuncVar := "SS1_A6_16DI_DI_Vars".DI16.cFuncVar);
END_REGION
END_FUNCTION
